PROGRAM PRG_TEST
VAR
    fb_AtPositionState_Test: FB_AtPositionState_Test;
    fb_AxisParameterSetExposed_Test: FB_AxisParameterSetExposed_Test;
    fb_MiscStatesErrorFFO_Test: FB_MiscStatesErrorFFO_Test;
    fb_MotionBPTM_Test: FB_MotionBPTM_Test;
    fb_MotionClearAsserts_Test: FB_MotionClearAsserts_Test;
    fb_MotionReadPMPSDBND_Test: FB_MotionReadPMPSDBND_Test;
    fbMotionVirtualFrameTest: FB_MotionVirtualFrame_Test;
    fb_TestHelperSetAndMove_Test: FB_TestHelperSetAndMove_Test;
    fb_PositionStateRead_Test: FB_PositionStateRead_Test;
    fb_PositionStateReadND_Test: FB_PositionStateReadND_Test;
    fb_PositionStateMove_Test: FB_PositionStateMove_Test;
    fb_PositionStateMoveND_Test: FB_PositionStateMoveND_Test;
    fb_PositionStateND_Test: FB_PositionStateND_Test;
    fb_NCErrorFFO_Test: FB_NCErrorFFO_Test;
    fb_StatePMPSEnables_Test: FB_StatePMPSEnables_Test;
    fb_PerMotorFFOND_Test: FB_PerMotorFFOND_Test;
    fb_StatePMPSEnablesND_Test: FB_StatePMPSEnablesND_Test;
    fb_PositionStatePMPSND_Test: FB_PositionStatePMPSND_Test;
    fb_StateSetupHelper_Test: FB_StateSetupHelper_Test;
    fb_TestStateInitTiming: FB_TestStateInitTiming;
    fb_PowerEnableMode_Test: FB_PowerEnableMode_Test;
    fb_MotionBacklashCompensation_Test: FB_MotionBacklashCompensation_Test;
    fb_MCS2DriveManager_Test: FB_MCS2DriveManager_Test;
END_VAR


TcUnit.RUN();

END_PROGRAM

(* stored: Version 1.1.0.1
   POU PRG_TEST: Id {4ab956a8-55df-43df-b997-1651a293eed5}, SpecialFunc None *)
